// TIA Portal V20 export
TYPE "LBP_typeMcp310PnInput"
TITLE = MCP 310 PN image / Image du MCP 310 PN
// Input image of MCP 310 PN / Image d'entrée du MCP 310 PN
   STRUCT
      standard { S7_SetPoint := 'True'} : "LBP_typeMcp310StandardInput";   // Input image of MCP 310 / Image d'entrée du MCP 310
      directKey1 : Bool;   // DT1
      directKey2 : Bool;   // DT2
      directKey3 : Bool;   // DT3
      directKey4 : Bool;   // DT4
      directKey5 : Bool;   // DT5
      directKey6 : Bool;   // DT6
      directKey7 : Bool;   // DT7
      directKey8 : Bool;   // DT8
      directKey9 : Bool;   // DT9
      directKey10 : Bool;   // DT10
      directKey11 : Bool;   // DT11
      directKey12 : Bool;   // DT12
      directKey13 : Bool;   // DT13
      directKey14 : Bool;   // DT14
      directKey15 : Bool;   // DT15
      directKey16 : Bool;   // DT16
      optionalKey1 : Bool;   // KT-IN1
      optionalKey2 : Bool;   // KT-IN2
      optionalKey3 : Bool;   // KT-IN3
      optionalKey4 : Bool;   // KT-IN4
      optionalKey5 : Bool;   // KT-IN5
      optionalKey6 : Bool;   // KT-IN6
      optionalKey7 : Bool;   // KT-IN7
      optionalKey8 : Bool;   // KT-IN8
      optionalKey9 : Bool;   // KT-IN9
      reserved111 : Bool;
      reserved112 : Bool;
      reserved113 : Bool;
      reserved114 : Bool;
      reserved115 : Bool;
      reserved116 : Bool;
      reserved117 : Bool;
      reserved12 : Byte;
      spindleOvrA : Bool;
      spindleOvrB : Bool;
      spindleOvrC : Bool;
      spindleOvrD : Bool;
      spindleOvrE : Bool;
      reserved135 : Bool;
      reserved136 : Bool;
      reserved137 : Bool;
   END_STRUCT;
END_TYPE
